Yaskawa INFORM job: SCIANA_MASTER_NOWY2.JBI

/JOB
//NAME SCIANA_MASTER_NOWY2
///FOLDERNAME KRIS-SCIANA
//POS
///NPOS 28,28,28,0,0,0
///TOOL 0
///POSTYPE PULSE
///PULSE
C00000=5012,38781,33405,-3737,88219,85582
C00001=5012,38781,33405,-3737,88219,85582
C00002=-13644,-92138,-120638,38655,87204,86250
C00003=-3569,-156345,-136276,3738,37668,81358
C00004=-97801,-92951,-68020,-42573,91743,12282
C00005=26932,41391,-30369,6536,105272,62664
C00006=147750,-31965,-71698,11557,98758,54427
C00007=228978,-94429,-102106,11557,98758,-20434
C00008=-41954,-92357,-91931,-694,81235,59832
C00009=19143,-90916,-90036,-16768,72453,41097
C00010=13148,3851,-75147,6736,62300,60674
C00011=-19622,89382,57086,542,94739,-201
C00012=3857,107043,326,1084,102018,80372
C00013=20488,129728,35048,-15297,94679,79335
C00014=26752,116740,10365,-10832,101628,84944
C00015=-2671,-162464,-131023,2021,-23223,-27872
C00016=-2671,-31387,-56562,2021,-23223,78061
C00017=7457,87076,9494,-2565,14741,80731
C00018=55255,-144335,-106474,-27033,-7250,-4370
C00019=-103661,-99969,-80124,-3650,-16231,-78554
C00020=-70468,-49830,-80124,-3650,74475,-78554
C00021=-17809,49263,-16328,-8127,84919,7903
C00022=16466,126359,28804,-9196,95410,70399
C00023=-81306,48778,44206,-5078,2277,-55818
C00024=-38214,88184,6233,-6392,80873,-25598
C00025=13601,139157,41546,-12188,94395,85883
C00026=29960,140181,41546,-12188,94395,86333
C00027=-314,141403,44956,-13517,93771,87051
BC00000=61339,583433,859490
BC00001=61339,583433,859490
BC00002=194821,433358,1073901
BC00003=85972,554727,117900
BC00004=365145,1359,801155
BC00005=165105,11813,1033268
BC00006=337965,17193,1016408
BC00007=337965,17193,1016408
BC00008=294910,15771,909310
BC00009=344649,733,1067002
BC00010=4442,187529,1013854
BC00011=150460,64597,1052617
BC00012=125260,23786,1075157
BC00013=137052,81055,1075158
BC00014=125260,578,1075157
BC00015=234035,34,1075174
BC00016=4525,66,1075174
BC00017=1047,287,1075169
BC00018=395584,33331,1067589
BC00019=390854,16,1053735
BC00020=396159,16,1053735
BC00021=333980,319,1064967
BC00022=135177,789,1073259
BC00023=398094,17,1057319
BC00024=309155,202,1060615
BC00025=125260,780,1075157
BC00026=65304,25846,1075157
BC00027=68533,631911,1075157
EC00000=0,0
EC00001=0,0
EC00002=-798147,556474
EC00003=-1,0
EC00004=0,0
EC00005=-1,0
EC00006=-1,0
EC00007=-1,0
EC00008=-1,0
EC00009=798156,0
EC00010=620788,-556477
EC00011=-620788,-556475
EC00012=0,-556476
EC00013=0,0
EC00014=798157,556476
EC00015=1596314,0
EC00016=1596314,0
EC00017=1596314,0
EC00018=1596314,1112952
EC00019=1596314,1112952
EC00020=1596314,1112952
EC00021=1596314,1112952
EC00022=1596314,1112952
EC00023=1596314,1112952
EC00024=1596314,1112952
EC00025=1596314,1112952
EC00026=1152894,-556476
EC00027=0,0
//INST
///DATE 2023/12/20 15:46
///ATTR SC,RW
///GROUP1 RB1,BS1
///GROUP2 ST1
NOP
'ZEROWANIE
'ZEROWANIE
'ZEROWANIE
DOUT OG#(198) 0
WAIT IG#(198)=0
DOUT OG#(200) 0
WAIT IG#(200)=0
MOVJ C00000 BC00000 VJ=40.00  +MOVJ EC00000 VJ=100.00
COMM JUMP *KAMERA
MOVJ C00001 BC00001 VJ=40.00  +MOVJ EC00001 VJ=100.00
COMM CALL JOB:GET_CAMERA
CALL JOB:0_-90
CALL JOB:R1_W01(KAMERA)(0,-90)
CALL JOB:125_90
CALL JOB:R1_W12(125,90)(KAMERA)
CALL JOB:-90_90
DOUT OG#(198) 100
WAIT IG#(198)=100
CALL JOB:R1_W26(-90,90)(KAMERA)
DOUT OG#(198) 101
WAIT IG#(198)=101
CALL JOB:R1_W23(-90,90)(KAMERA)KM-OK
DOUT OG#(198) 102
WAIT IG#(198)=102
MOVJ C00002 BC00002 VJ=30.00  +MOVJ EC00002 VJ=40.00
MOVJ C00003 BC00003 VJ=30.00  +MOVJ EC00003 VJ=40.00
COMM CALL JOB:LEAVE_CAMERA
'KONIEC SPAWANIA ZE SLEDZENIEM
'KAMERA SERVO ROBOT
'----------------------
*KAMERA
CALL JOB:CLEAN-R1_LONG
DOUT OG#(198) 103
WAIT IG#(198)=103
CALL JOB:0_0
MOVJ C00004 BC00004 VJ=30.00  +MOVJ EC00004 VJ=40.00
DOUT OG#(198) 1
WAIT IG#(198)=1
CALL JOB:R1_W03,5,7(0,0)OK-KM
DOUT OG#(198) 2
WAIT IG#(198)=2
CALL JOB:CLEAN-R1_LONG
MOVJ C00005 BC00005 VJ=20.00  +MOVJ EC00005 VJ=40.00
MOVJ C00006 BC00006 VJ=20.00  +MOVJ EC00006 VJ=40.00
MOVJ C00007 BC00007 VJ=20.00  +MOVJ EC00007 VJ=40.00
DOUT OG#(198) 3
WAIT IG#(198)=3
CALL JOB:R1_W14,16(0,0)OK-KM
CALL JOB:CLEAN-R1_LONG
MOVJ C00008 BC00008 VJ=20.00  +MOVJ EC00008 VJ=40.00
DOUT OG#(198) 5
WAIT IG#(198)=5
CALL JOB:R1_W17,20,22(0,0)OK-KM
CALL JOB:CLEAN-R1_LONG
CALL JOB:R1_W30(0,0)OK-KM
CALL JOB:CLEAN-R1_LONG
DOUT OG#(198) 9
WAIT IG#(198)=9
CALL JOB:R1_W33(0,0)KM-OK
DOUT OG#(198) 10
WAIT IG#(198)=10
'----------------------
'231112OKAW
'SPAWANIE DLA POZYCJI 90_0
CALL JOB:90_0
DOUT OG#(198) 11
WAIT IG#(198)=11
MOVJ C00009 BC00009 VJ=20.00  +MOVJ EC00009 VJ=40.00
CALL JOB:CLEAN-R1_LONG
CALL JOB:R1_W27-A3(90,0)OK-KM
CALL JOB:CLEAN-R1_LONG
CALL JOB:R1_W27-A5(90,0)OK-KM
CALL JOB:CLEAN-R1_LONG
DOUT OG#(198) 15
WAIT IG#(198)=15
CALL JOB:R1_W35-36-A2(90,0)KM-OK
CALL JOB:CLEAN-R1_LONG
CALL JOB:R1_W45-48(90,0)KM-OK
DOUT OG#(198) 18
WAIT IG#(198)=18
'---------------------
'AWOK
'SPAWANIE DLA POZYCJI 70_-90
CALL JOB:70_-90
MOVJ C00010 BC00010 VJ=20.00  +MOVJ EC00010 VJ=100.00
DOUT OG#(198) 19
WAIT IG#(198)=19
CALL JOB:CLEAN-R1_LONG
DOUT OG#(198) 20
WAIT IG#(198)=20
CALL JOB:R1_W27-A2(70,-90)OK-KM
DOUT OG#(198) 21
WAIT IG#(198)=21
'---------------------
'ZMIANA POZYCJI SPAWANIA -70_-90
'AWOK
CALL JOB:-70_-90
DOUT OG#(198) 22
WAIT IG#(198)=22
MOVJ C00011 BC00011 VJ=20.00  +MOVJ EC00011 VJ=40.00
CALL JOB:CLEAN-R1_LONG
DOUT OG#(198) 23
WAIT IG#(198)=23
CALL JOB:R1_W09,10(-70,-90)
CALL JOB:CLEAN-R1_LONG
CALL JOB:R1_W66-67(-70,-90)KM-OK
DOUT OG#(198) 26
WAIT IG#(198)=26
'---------------------
'AWOK
'ZMIANA POZYCJI SPAWANIA -90_-90
CALL JOB:-90_-90
DOUT OG#(198) 27
WAIT IG#(198)=27
CALL JOB:CLEAN-R1_LONG
CALL JOB:R1_W68-69(-90,-90)KM-OK
CALL JOB:CLEAN-R1_LONG
CALL JOB:R1_W70(-90,-90)KM-OK
DOUT OG#(198) 30
WAIT IG#(198)=30
'ZMIANA POZYCJI SPAWANIA -45_-90
'AWOK
CALL JOB:-45_-90
DOUT OG#(198) 31
WAIT IG#(198)=31
CALL JOB:CLEAN-R1_LONG
DOUT OG#(198) 32
WAIT IG#(198)=32
CALL JOB:R1_W72(-45,-90)KM-OK
DOUT OG#(198) 33
WAIT IG#(198)=33
'ZMIANA POZYCJI SPAWANIA 0_-90
CALL JOB:0_-90
DOUT OG#(198) 34
WAIT IG#(198)=34
MOVJ C00012 BC00012 VJ=20.00  +MOVJ EC00012 VJ=30.00
CALL JOB:CLEAN-R1_LONG
DOUT OG#(198) 35
WAIT IG#(198)=35
CALL JOB:R1_W73(0,-90)KM-OK
DOUT OG#(198) 36
WAIT IG#(198)=36
'ZMIANA POZYCJI SPAWANIA 0_0
'AWOK
CALL JOB:0_0
DOUT OG#(198) 37
WAIT IG#(198)=37
MOVJ C00013 BC00013 VJ=20.00  +MOVJ EC00013 VJ=30.00
CALL JOB:CLEAN-R1_LONG
DOUT OG#(198) 38
WAIT IG#(198)=38
CALL JOB:R1_W60,62(0,0)KM-OK
CALL JOB:CLEAN-R1_LONG
CALL JOB:R1_72,2(0,0)KM-OK
DOUT OG#(198) 39
WAIT IG#(198)=39
'ZMIANA POZYCJI SPAWANIA 80_0
CALL JOB:80_0
DOUT OG#(198) 40
WAIT IG#(198)=40
CALL JOB:CLEAN-R1_LONG
CALL JOB:R1_W43-44-A1(80,0))KM-OK
DOUT OG#(198) 42
WAIT IG#(198)=42
'ZMIANA POZYCJI SPAWANIA 90_90
'AWOK
CALL JOB:90_90
DOUT OG#(198) 43
WAIT IG#(198)=43
MOVJ C00014 BC00014 VJ=20.00  +MOVJ EC00014 VJ=30.00
CALL JOB:CLEAN-R1_LONG
DOUT OG#(198) 44
WAIT IG#(198)=44
CALL JOB:R1_W49-52-A2(90,90)KM-OK
DOUT OG#(198) 45
WAIT IG#(198)=45
'ZMIANA POZYCJI SPAWANIA 90_180
'AWOK
CALL JOB:90_180
DOUT OG#(198) 46
WAIT IG#(198)=46
CALL JOB:CLEAN-R1_LONG
CALL JOB:R1_W27-A4(90,180)KM-OK
CALL JOB:CLEAN-R1_LONG
CALL JOB:R1_W35-36-A1(90,180)KM-OK
CALL JOB:CLEAN-R1_LONG
CALL JOB:R1_W49-52-A1(90,180)KM-OK
DOUT OG#(198) 52
WAIT IG#(198)=52
'AWOK
'ZMIANA POZYCJI SPAWANIA 80_180
CALL JOB:80_180
DOUT OG#(198) 53
WAIT IG#(198)=53
CALL JOB:CLEAN-R1_LONG
DOUT OG#(198) 54
WAIT IG#(198)=54
CALL JOB:R1_W43-44-A2(80,180)KM-OK
'ZMIANA POZYCJI SPAWANIA 180_0
'AWOK
DOUT OG#(198) 55
WAIT IG#(198)=55
CALL JOB:180_0
DOUT OG#(198) 56
WAIT IG#(198)=56
MOVJ C00015 BC00015 VJ=20.00  +MOVJ EC00015 VJ=100.00
MOVJ C00016 BC00016 VJ=20.00  +MOVJ EC00016 VJ=100.00
MOVJ C00017 BC00017 VJ=20.00  +MOVJ EC00017 VJ=100.00
CALL JOB:CLEAN-R1_LONG
CALL JOB:R1_W49-52-A5(180,0)KM-OK
DOUT OG#(198) 58
WAIT IG#(198)=58
'ZMIANA POZYCJI SPAWANIA 180_180
CALL JOB:180_180
DOUT OG#(198) 59
WAIT IG#(198)=59
MOVJ C00018 BC00018 VJ=20.00  +MOVJ EC00018 VJ=100.00
MOVJ C00019 BC00019 VJ=20.00  +MOVJ EC00019 VJ=100.00
MOVJ C00020 BC00020 VJ=20.00  +MOVJ EC00020 VJ=100.00
MOVJ C00021 BC00021 VJ=20.00  +MOVJ EC00021 VJ=100.00
MOVJ C00022 BC00022 VJ=20.00  +MOVJ EC00022 VJ=100.00
CALL JOB:CLEAN-R1_LONG
CALL JOB:R1_W28-29-A1(180,180)KM-OK
DOUT OG#(198) 63
WAIT IG#(198)=63
' POZYCJI BEZ ZMIAN -180_180
MOVJ C00023 BC00023 VJ=20.00  +MOVJ EC00023 VJ=100.00
MOVJ C00024 BC00024 VJ=20.00  +MOVJ EC00024 VJ=100.00
MOVJ C00025 BC00025 VJ=20.00  +MOVJ EC00025 VJ=100.00
CALL JOB:CLEAN-R1_LONG
CALL JOB:R1_W27-A6(-180,180)KM-OK
DOUT OG#(198) 65
WAIT IG#(198)=65
'ZMIANA POZYCJI SPAWANIA 130_-90
CALL JOB:130_-90
DOUT OG#(198) 66
WAIT IG#(198)=66
MOVJ C00026 BC00026 VJ=20.00  +MOVJ EC00026 VJ=100.00
CALL JOB:CLEAN-R1_LONG
CALL JOB:R1_W63-A2(130,-90)(JEDENR)KM-OK
'ZMIANA POZYCJI SPAWANIA 120_-90
CALL JOB:120_-90
DOUT OG#(198) 68
WAIT IG#(198)=68
CALL JOB:CLEAN-R1_LONG
DOUT OG#(198) 69
WAIT IG#(198)=69
CALL JOB:R1_W63-A1(120,-90)KM-OK
DOUT OG#(198) 70
WAIT IG#(198)=70
CALL JOB:0_0
'SZCZEPIANIE BATMANA I BOCZKOW
PAUSE
PAUSE
PAUSE
CALL JOB:-70_-90
CALL JOB:R1_BATVER2(-70,-90)KM-OK
PAUSE
DOUT OG#(198) 71
WAIT IG#(198)=71
CALL JOB:-70_-90
DOUT OG#(198) 72
WAIT IG#(198)=72
CALL JOB:0_0
MOVJ C00027 BC00027 VJ=40.00  +MOVJ EC00027 VJ=40.00
'ZEROWANIE
'ZEROWANIE
'ZEROWANIE
DOUT OG#(200) 0
WAIT IG#(200)=0
DOUT OG#(198) 0
WAIT IG#(198)=0
END
